FUNCTION_BLOCK EBSlave2181 (* Service Interface Function Block Type *)
  (* Description: Copyright (c) 2016 fortiss GmbH This program and the accompanying materials are made available under the terms of the Eclipse Public License 2.0 which is available at https://www.eclipse.org/legal/epl-2.0/ SPDX-License-Identifier: EPL-2.0 *)
  (* Version 1.0, 2016-11-30, Johannes Messmer, fortiss GmbH *)
  (* Version 3.0, 2025-04-14, Patrick Aigner, changed package *)
  PACKAGE eclipse4diac::io::embrick;
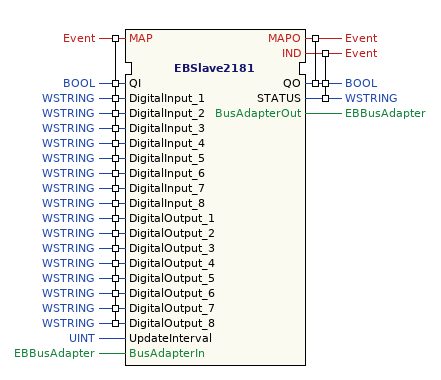
  EVENT_INPUT
    MAP WITH DigitalInput_1, DigitalInput_2, DigitalInput_5, DigitalInput_3, DigitalInput_4, DigitalInput_6, DigitalInput_7, DigitalInput_8, DigitalOutput_1, DigitalOutput_2, DigitalOutput_3, DigitalOutput_4, DigitalOutput_5, DigitalOutput_6, DigitalOutput_7, DigitalOutput_8, QI; (* Map Pins *)
  END_EVENT
  EVENT_OUTPUT
    MAPO WITH QO; (* Confirm Pin Mapping *)
    IND WITH QO, STATUS; (* Indication from Resource *)
  END_EVENT
  VAR_INPUT
    QI : BOOL; (* Event Input Qualifier *)
    DigitalInput_1 : WSTRING;
    DigitalInput_2 : WSTRING;
    DigitalInput_3 : WSTRING;
    DigitalInput_4 : WSTRING;
    DigitalInput_5 : WSTRING;
    DigitalInput_6 : WSTRING;
    DigitalInput_7 : WSTRING;
    DigitalInput_8 : WSTRING;
    DigitalOutput_1 : WSTRING;
    DigitalOutput_2 : WSTRING;
    DigitalOutput_3 : WSTRING;
    DigitalOutput_4 : WSTRING;
    DigitalOutput_5 : WSTRING;
    DigitalOutput_6 : WSTRING;
    DigitalOutput_7 : WSTRING;
    DigitalOutput_8 : WSTRING;
    UpdateInterval : UINT; (* Update interval of slave module in Hz (inherited from Master) *)
  END_VAR
  VAR_OUTPUT
    QO : BOOL; (* Event Output Qualifier *)
    STATUS : WSTRING; (* Service Status *)
  END_VAR
  SOCKETS
    BusAdapterIn : eclipse4diac::io::embrick::EBBusAdapter;
  END_SOCKETS
  PLUGS
    BusAdapterOut : eclipse4diac::io::embrick::EBBusAdapter;
  END_PLUGS
END_FUNCTION_BLOCK
